FUNCTION_BLOCK CyclicEventDetection
VAR_INPUT
END_VAR
VAR_OUTPUT
END_VAR
VAR
  message_counter: INT;
  event_counter: INT;
  messages: ARRAY[1..Properties.NUM_CYCLIC_DETECTION_MESSAGES] OF ST_CyclicMessageDetection;
  events: ARRAY[1..Properties.NUM_EVENTS] OF ST_CyclicEventDetection;
END_VAR

METHOD PRIVATE dec_event_counter
VAR_INPUT
END_VAR
event_counter := LIMIT(0, event_counter - 1, Properties.NUM_EVENTS);
END_METHOD

METHOD PRIVATE reset_event
VAR_INPUT
  index: INT;
END_VAR
events[index].submitted_in_last_invocation := FALSE;
END_METHOD

METHOD PRIVATE activate_event
VAR_INPUT
  index: INT;
END_VAR
events[index].submitted_in_last_invocation := TRUE;
END_METHOD

METHOD PRIVATE activate_message
VAR_INPUT
  index: INT;
END_VAR
messages[index].message_submitted := TRUE;
END_METHOD

METHOD PRIVATE dec_message_counter
VAR_INPUT
END_VAR
message_counter := LIMIT(0, message_counter - 1, Properties.NUM_CYCLIC_DETECTION_MESSAGES);
END_METHOD

METHOD PRIVATE reset_message
VAR_INPUT
  index: INT;
END_VAR
messages[index].message_submitted := FALSE;
END_METHOD

METHOD PUBLIC reset_messages
VAR_INPUT
END_VAR
VAR
  i: INT;
END_VAR
FOR i:=1 TO message_counter DO
  reset_message(i);
END_FOR
END_METHOD

METHOD PRIVATE message_index_valid : BOOL
VAR_INPUT
  index: INT;
END_VAR
message_index_valid := (1 <= index) AND (index <= Properties.NUM_CYCLIC_DETECTION_MESSAGES);
END_METHOD

METHOD PUBLIC reactivate_event
VAR_INPUT
  index: INT;
END_VAR
IF event_id_valid(index) THEN
  activate_event(index);
END_IF
END_METHOD

METHOD PUBLIC get_event_index : INT
VAR_INPUT
  id: INT;
END_VAR
VAR
  i: INT;
END_VAR
FOR i:=1 TO event_counter DO
  IF events[i].id = id THEN
    get_event_index := i;
    EXIT;
  END_IF
END_FOR
END_METHOD

METHOD PUBLIC event_was_called_in_last_invocation : BOOL
VAR_INPUT
  id: INT;
END_VAR
VAR
  i: INT;
END_VAR
FOR i:=1 TO event_counter DO
  IF events[i].id = id THEN
    event_was_called_in_last_invocation := TRUE;
    EXIT;
	END_IF
END_FOR
END_METHOD

METHOD PRIVATE inc_event_counter
VAR_INPUT
END_VAR
event_counter := LIMIT(1, event_counter + 1, Properties.NUM_EVENTS);
END_METHOD

METHOD PUBLIC reset_events
VAR_INPUT
END_VAR
VAR
  i: INT;
END_VAR
FOR i:=1 TO event_counter DO
  reset_event(i);
END_FOR
END_METHOD

METHOD PRIVATE remove_deactivated_messages
VAR_INPUT
END_VAR
VAR
  i: INT;
  filldata: ST_CyclicMessageDetection;
END_VAR
FOR i:=1 TO message_counter DO
  IF NOT messages[i].message_submitted THEN
    remove_field_from_array(
      index_to_remove:=i,
      size_filldata:=SIZEOF(filldata),
      adr_filldata:=ADR(filldata),
      size_memory_buffer:=SIZEOF(messages),
      adr_memory_buffer:=ADR(messages)
    );
    dec_message_counter();
    i := i - 1;
	END_IF
END_FOR
END_METHOD

METHOD PRIVATE remove_deactivated_events
VAR_INPUT
END_VAR
VAR
  i: INT;
  filldata: ST_CyclicEventDetection;
END_VAR
FOR i:=1 TO event_counter DO
  IF NOT events[i].submitted_in_last_invocation THEN
    remove_field_from_array(
      index_to_remove:=i,
      size_filldata:=SIZEOF(filldata),
      adr_filldata:=ADR(filldata),
      size_memory_buffer:=SIZEOF(events),
      adr_memory_buffer:=ADR(events)
    );
    dec_event_counter();
    i := i - 1;
	END_IF
END_FOR
END_METHOD

METHOD PUBLIC add_message
VAR_INPUT
  ev: EventMessage;
END_VAR
VAR
  event_index: INT;
END_VAR
IF NOT max_number_events_reached() THEN
  inc_message_counter();
  messages[message_counter].ev := ev;
  activate_message(message_counter);
END_IF
END_METHOD

METHOD get_message_index : INT
VAR_IN_OUT
  ev: EventMessage;
END_VAR
VAR
  i: INT;
END_VAR
FOR i:=1 TO message_counter DO
  IF messages[i].ev.message.str = ev.message.str THEN
    get_message_index := i;
    EXIT;
  END_IF
END_FOR
END_METHOD

METHOD PRIVATE max_number_events_reached : BOOL
VAR_INPUT
END_VAR
max_number_events_reached := message_counter >= Properties.NUM_CYCLIC_DETECTION_MESSAGES;
END_METHOD

METHOD PRIVATE event_id_valid : BOOL
VAR_INPUT
  id: INT;
END_VAR
event_id_valid := (1 <= id) AND (id <= Properties.NUM_EVENTS);
END_METHOD

METHOD PUBLIC cyclic_call
VAR_INPUT
END_VAR
remove_deactivated_events();
remove_deactivated_messages();
reset_events();
reset_messages();
END_METHOD

METHOD PRIVATE inc_message_counter
VAR_INPUT
END_VAR
message_counter := LIMIT(1, message_counter + 1, Properties.NUM_CYCLIC_DETECTION_MESSAGES);
END_METHOD

METHOD PUBLIC reactivate_message
VAR_INPUT
  index: INT;
END_VAR
IF event_id_valid(index) THEN
  activate_message(index);
END_IF
END_METHOD

METHOD PUBLIC add_event
VAR_INPUT
  id: INT;
END_VAR
VAR
  event_index: INT;
END_VAR
inc_event_counter();
events[event_counter].id := id;
activate_event(event_counter);
END_METHOD

END_FUNCTION_BLOCK

(* stored: Version 1.1.0.1, ProductVersion 3.1.4022.18
   POU CyclicEventDetection: Id {1c97c1bd-572d-44e9-8e88-b7c37ccb1356}, SpecialFunc None
   Method dec_event_counter: Id {0784a32d-3d83-4525-8c5d-be6debc405ce}
   Method reset_event: Id {0a70bd33-007f-4294-8a73-d10e283a42ce}
   Method activate_event: Id {0f0242e9-5189-4722-8245-48fde68885c7}
   Method activate_message: Id {11dcbf06-b87b-40e3-a22c-1322dcf8d3ab}
   Method dec_message_counter: Id {39864b04-eef3-41d8-b15c-b9ce24cdcb1a}
   Method reset_message: Id {3ab35474-895f-41ca-8f7f-b48ddc7ca55d}
   Method reset_messages: Id {58053604-4b09-40fa-ae5a-6a335837d9df}
   Method message_index_valid: Id {7195b9d5-9c83-49b2-8210-1747bbb58eb4}
   Method reactivate_event: Id {7220f904-f441-4eff-b09b-5bb0b53619c6}
   Method get_event_index: Id {74a71643-ecf3-4bf5-9113-b1d0b8e41be8}
   Method event_was_called_in_last_invocation: Id {792ac793-573f-480e-9aac-6f74d8eb6b0f}
   Method inc_event_counter: Id {7bd905bd-b8a4-4f50-9ee7-d0fba39c52a1}
   Method reset_events: Id {7fc3b6d4-9905-410c-be29-b8c70d0b9bdf}
   Method remove_deactivated_messages: Id {800606f0-f6b4-4f9b-989f-2c47c5a54588}
   Method remove_deactivated_events: Id {89efefac-cb81-46b4-8514-400dda4a7e5b}
   Method add_message: Id {98a044d6-bc69-4b90-8daf-4c89e29ec295}
   Method get_message_index: Id {a046a0fe-7a93-44d8-a74c-feebbbc6fcc6}
   Method max_number_events_reached: Id {b34f7417-8ca3-4515-960a-8ab7223c93f0}
   Method event_id_valid: Id {c41f610a-d0c9-4f62-9bf3-87bbda6a200b}
   Method cyclic_call: Id {c7bed164-f925-46cd-910a-bb07f34b0bbb}
   Method inc_message_counter: Id {d0c0bc51-8423-474b-8101-7c82bfc231c6}
   Method reactivate_message: Id {d16e9fda-f182-4b12-830f-8fd08512ff2c}
   Method add_event: Id {dbe32403-a802-4456-9932-b36bf1dfcc8a} *)
